{attribute 'Tc2GvlVarNames'}
VAR_GLOBAL

	(* MGMT_Zustand_Status *)
	E_MGMT_Zustand_Status_Idle_Sperre		: SINT := 0;
	E_MGMT_Zustand_Status_Betriebsbereit	: SINT := 1;
	E_MGMT_Zustand_Status_Betrieb			: SINT := 8;
	E_MGMT_Zustand_Status_Betrieb_Sperre	: SINT := 9;
	E_MGMT_Zustand_Status_Stoerung			: SINT := 99;

	(* MGMT_Zustand_Regelung_Modus *)
	E_MGMT_Regelung_Modus_Auto				: SINT := 0;
	E_MGMT_Regelung_Modus_T_Unten			: SINT := 1;
	E_MGMT_Regelung_Modus_T_Oben			: SINT := 2;


END_VAR

(* stored: Version 1.1.0.1, ProductVersion 3.1.4024.9
   GVL Con_MGMT: Id {3bb00c59-1932-46db-bcdb-2233549a3641} *)
